(* Schneider Machine Expert - Basic project Latihan VFD, file version 2.1.0.0 *)
(* ProjectInformations: Name=New project *)

HARDWARE
  Cpu 0: TM221ME16R/G
  EthernetConfiguration: NetworkName=M221, IpAllocationMode=FixedAddress, IpAddress=192.168.0.10, SubnetMask=255.255.255.0
  SerialLineConfiguration: Baud=Baud19200, Parity=ParityEven, DataBits=DataBits8, StopBits=StopBits1, PhysicalMedium=PhysicalMediumRs485, TransmissionMode=TransmissionModeModbusRtu, SlaveId=1, Addressing=SlaveAddressing
  MastTask: UsePeriodScanMode=false, PeriodScan=100
  FastTask: Period=255
  CpuBehavior: StartingMode=StartAsPreviousState, AutoSaveRamOnEeprom=true, WatchdogPeriod=250

SYMBOLS  (address, symbol, comment, settings)
  %I0.0     PB_1
  %I0.1     PB_2
  %Q0.0     L1
  %Q0.1     L3
  %Q0.2     L4
  %Q0.3     L5
  %IW0.0      [Type=Type_0_10V, Scope=Scope_Normal, Minimum=0, Maximum=1000]

POU New POU
  (* SectionNumber=1 *)

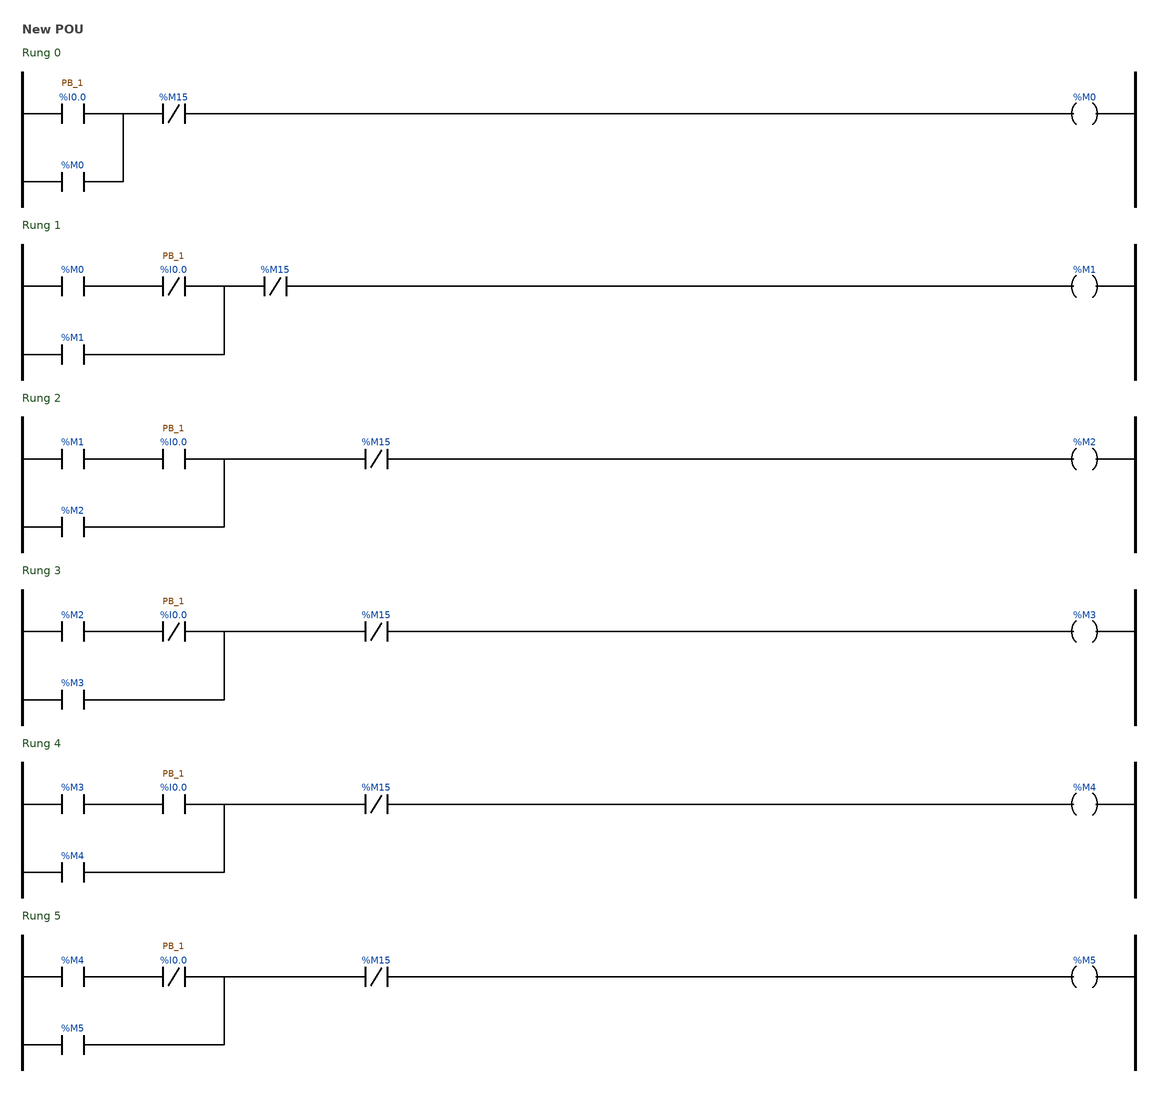

// Rung 0
  LD %I0.0                (* PB_1 *)
  OR %M0
  ANDN %M15
  ST %M0
  // as ST:
  //   %M0 := (PB_1 OR %M0) AND NOT %M15;

// Rung 1
  LD %M0
  ANDN %I0.0              (* PB_1 *)
  OR %M1
  ANDN %M15
  ST %M1
  // as ST:
  //   %M1 := (%M0 AND NOT PB_1 OR %M1) AND NOT %M15;

// Rung 2
  LD %M1
  AND %I0.0               (* PB_1 *)
  OR %M2
  ANDN %M15
  ST %M2
  // as ST:
  //   %M2 := (%M1 AND PB_1 OR %M2) AND NOT %M15;

// Rung 3
  LD %M2
  ANDN %I0.0              (* PB_1 *)
  OR %M3
  ANDN %M15
  ST %M3
  // as ST:
  //   %M3 := (%M2 AND NOT PB_1 OR %M3) AND NOT %M15;

// Rung 4
  LD %M3
  AND %I0.0               (* PB_1 *)
  OR %M4
  ANDN %M15
  ST %M4
  // as ST:
  //   %M4 := (%M3 AND PB_1 OR %M4) AND NOT %M15;

// Rung 5
  LD %M4
  ANDN %I0.0              (* PB_1 *)
  OR %M5
  ANDN %M15
  ST %M5
  // as ST:
  //   %M5 := (%M4 AND NOT PB_1 OR %M5) AND NOT %M15;

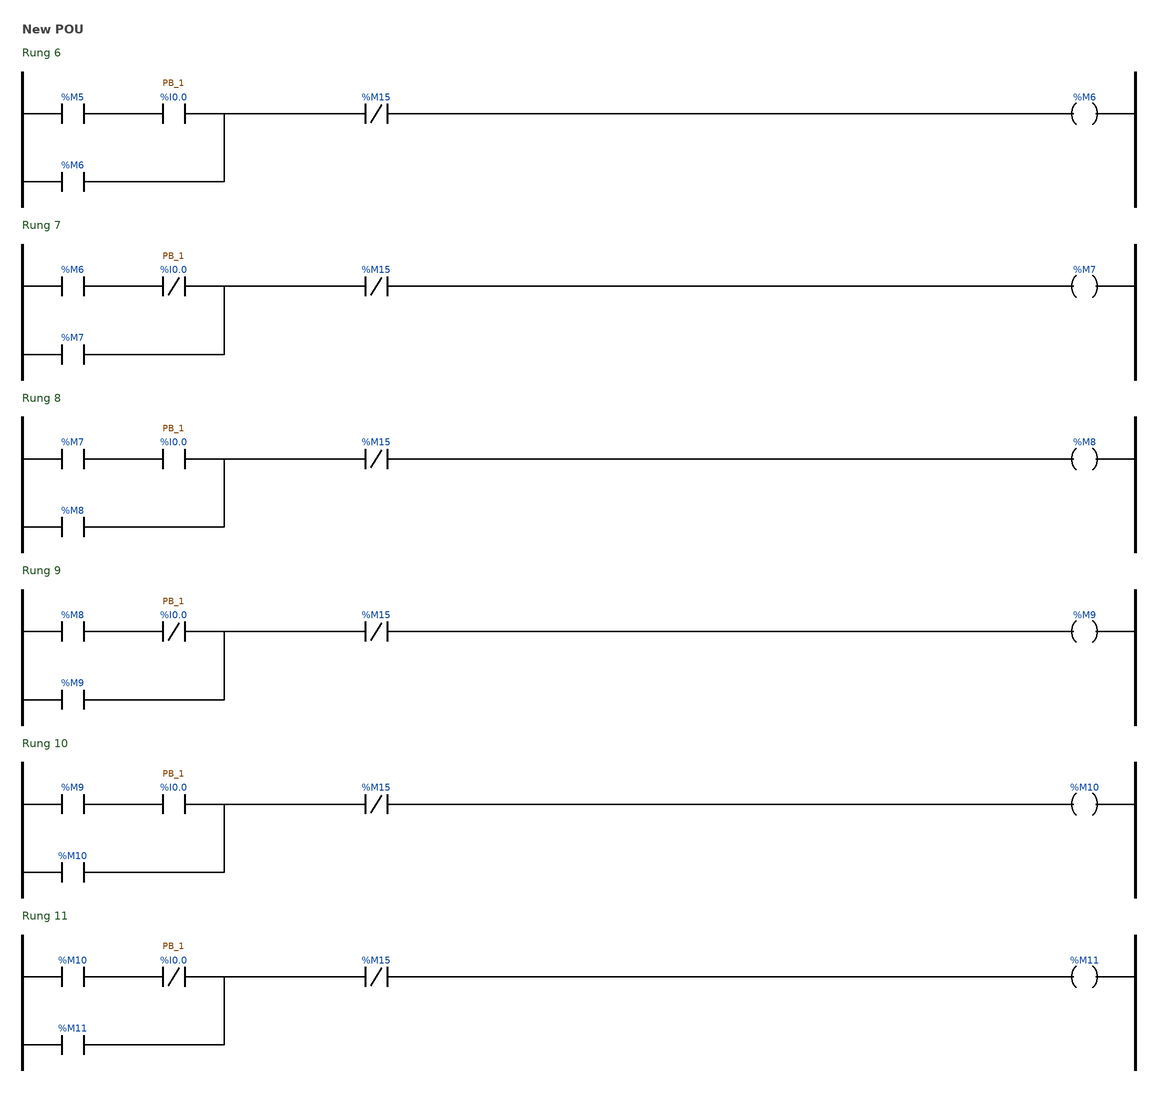

// Rung 6
  LD %M5
  AND %I0.0               (* PB_1 *)
  OR %M6
  ANDN %M15
  ST %M6
  // as ST:
  //   %M6 := (%M5 AND PB_1 OR %M6) AND NOT %M15;

// Rung 7
  LD %M6
  ANDN %I0.0              (* PB_1 *)
  OR %M7
  ANDN %M15
  ST %M7
  // as ST:
  //   %M7 := (%M6 AND NOT PB_1 OR %M7) AND NOT %M15;

// Rung 8
  LD %M7
  AND %I0.0               (* PB_1 *)
  OR %M8
  ANDN %M15
  ST %M8
  // as ST:
  //   %M8 := (%M7 AND PB_1 OR %M8) AND NOT %M15;

// Rung 9
  LD %M8
  ANDN %I0.0              (* PB_1 *)
  OR %M9
  ANDN %M15
  ST %M9
  // as ST:
  //   %M9 := (%M8 AND NOT PB_1 OR %M9) AND NOT %M15;

// Rung 10
  LD %M9
  AND %I0.0               (* PB_1 *)
  OR %M10
  ANDN %M15
  ST %M10
  // as ST:
  //   %M10 := (%M9 AND PB_1 OR %M10) AND NOT %M15;

// Rung 11
  LD %M10
  ANDN %I0.0              (* PB_1 *)
  OR %M11
  ANDN %M15
  ST %M11
  // as ST:
  //   %M11 := (%M10 AND NOT PB_1 OR %M11) AND NOT %M15;

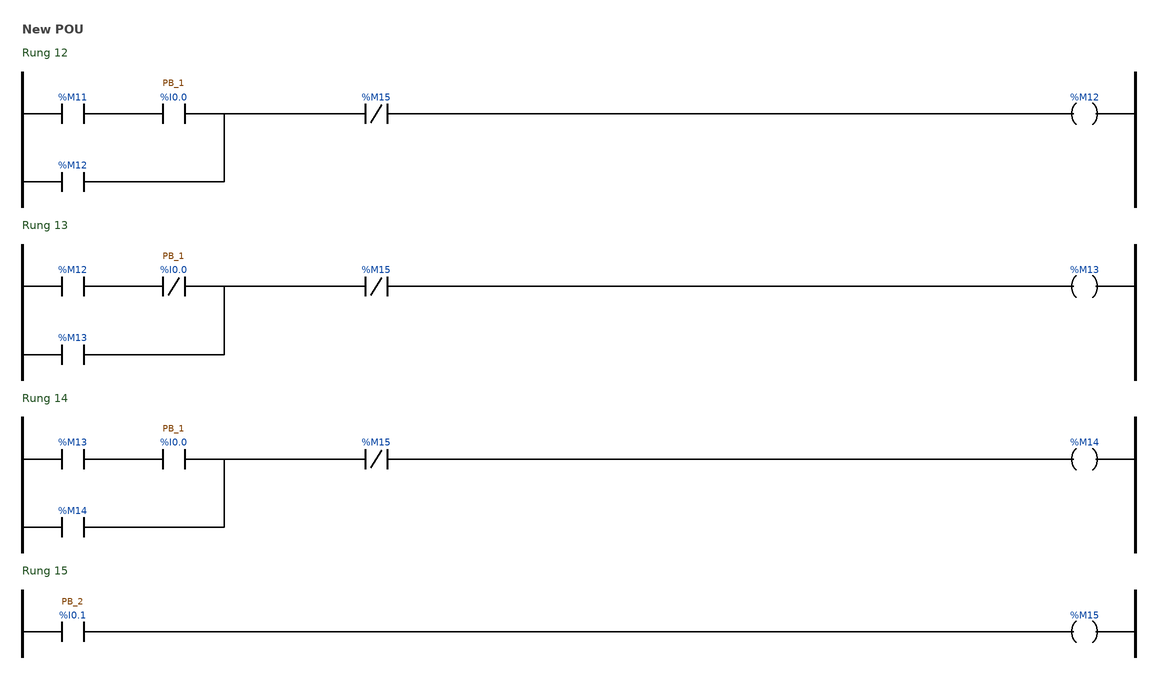

// Rung 12
  LD %M11
  AND %I0.0               (* PB_1 *)
  OR %M12
  ANDN %M15
  ST %M12
  // as ST:
  //   %M12 := (%M11 AND PB_1 OR %M12) AND NOT %M15;

// Rung 13
  LD %M12
  ANDN %I0.0              (* PB_1 *)
  OR %M13
  ANDN %M15
  ST %M13
  // as ST:
  //   %M13 := (%M12 AND NOT PB_1 OR %M13) AND NOT %M15;

// Rung 14
  LD %M13
  AND %I0.0               (* PB_1 *)
  OR %M14
  ANDN %M15
  ST %M14
  // as ST:
  //   %M14 := (%M13 AND PB_1 OR %M14) AND NOT %M15;

// Rung 15
  LD %I0.1                (* PB_2 *)
  ST %M15
  // as ST:
  //   %M15 := PB_2;

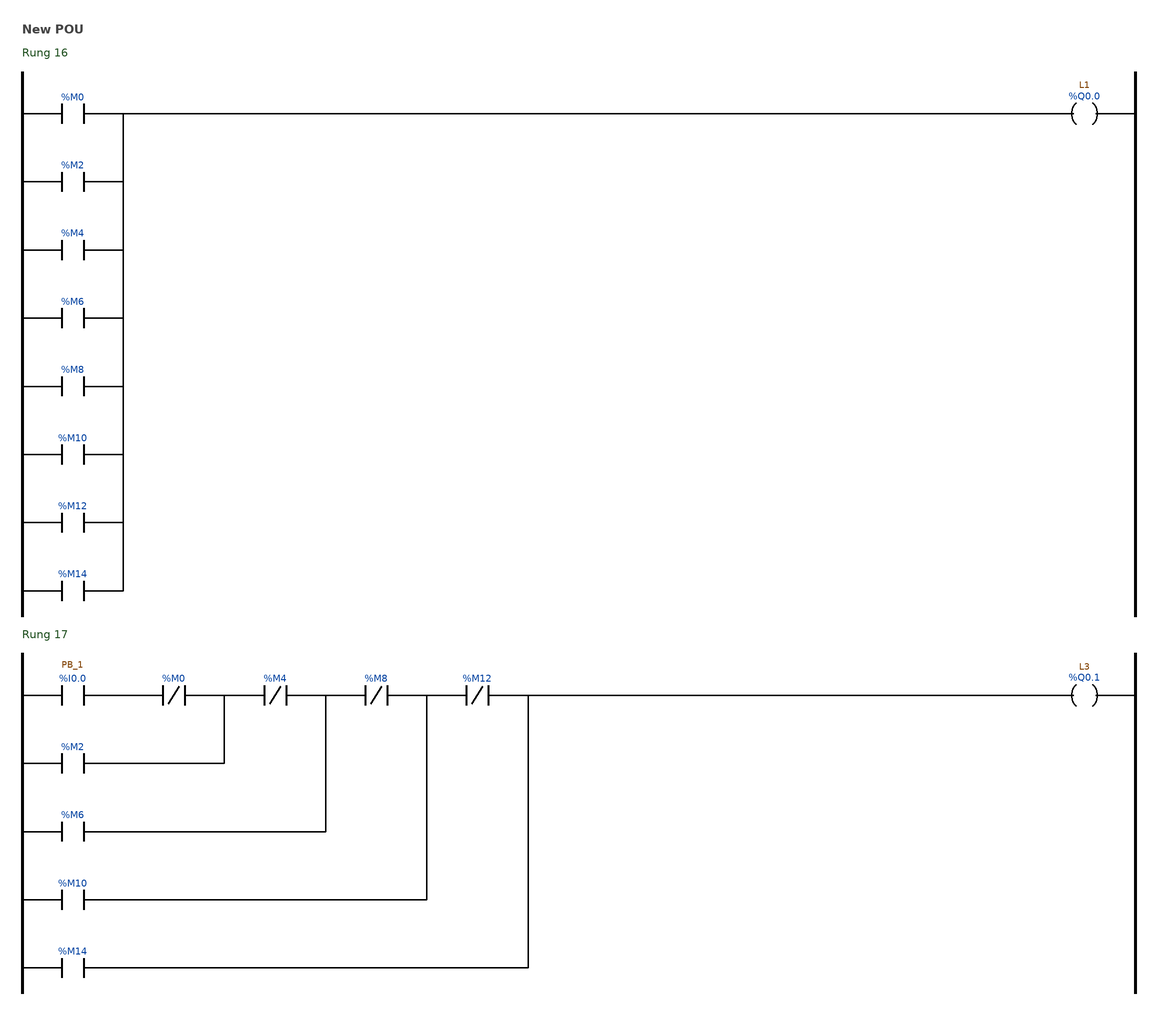

// Rung 16
  LD %M0
  OR %M2
  OR %M4
  OR %M6
  OR %M8
  OR %M10
  OR %M12
  OR %M14
  ST %Q0.0                (* L1 *)
  // as ST:
  //   L1 := %M0 OR %M2 OR %M4 OR %M6 OR %M8 OR %M10 OR %M12 OR %M14;

// Rung 17
  LD %I0.0                (* PB_1 *)
  ANDN %M0
  OR %M2
  ANDN %M4
  OR %M6
  ANDN %M8
  OR %M10
  ANDN %M12
  OR %M14
  ST %Q0.1                (* L3 *)
  // as ST:
  //   L3 := (((PB_1 AND NOT %M0 OR %M2) AND NOT %M4 OR %M6) AND NOT %M8 OR %M10) AND NOT %M12 OR %M14;

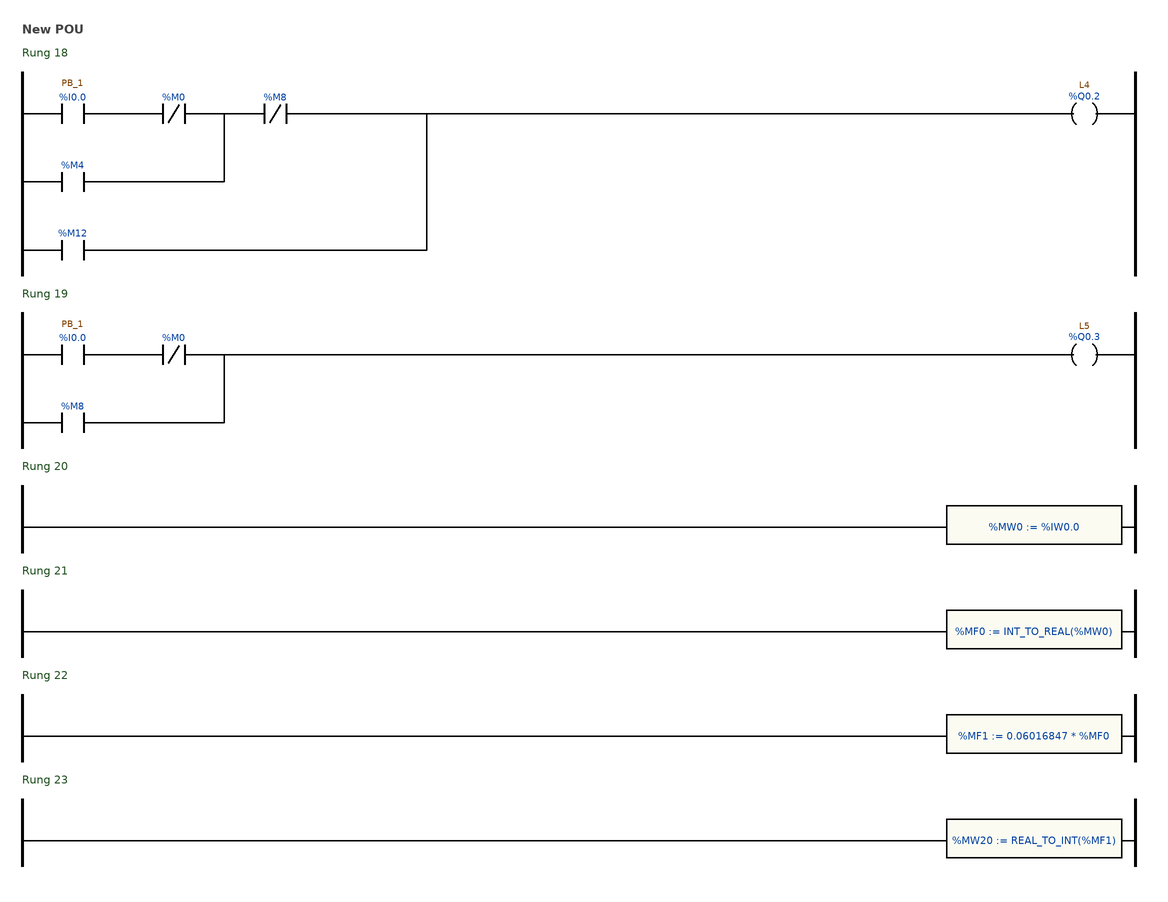

// Rung 18
  LD %I0.0                (* PB_1 *)
  ANDN %M0
  OR %M4
  ANDN %M8
  OR %M12
  ST %Q0.2                (* L4 *)
  // as ST:
  //   L4 := (PB_1 AND NOT %M0 OR %M4) AND NOT %M8 OR %M12;

// Rung 19
  LD %I0.0                (* PB_1 *)
  ANDN %M0
  OR %M8
  ST %Q0.3                (* L5 *)
  // as ST:
  //   L5 := PB_1 AND NOT %M0 OR %M8;

// Rung 20
  LD 1
  [ %MW0 := %IW0.0 ]
  // as ST:
  //   %MW0 := %IW0.0;

// Rung 21
  LD 1
  [ %MF0 := INT_TO_REAL ( %MW0 ) ]
  // as ST:
  //   %MF0 := INT_TO_REAL ( %MW0 );

// Rung 22
  LD 1
  [ %MF1 := 0.06016847 * %MF0 ]
  // as ST:
  //   %MF1 := 0.06016847 * %MF0;

// Rung 23
  LD 1
  [ %MW20 := REAL_TO_INT ( %MF1 ) ]
  // as ST:
  //   %MW20 := REAL_TO_INT ( %MF1 );
